PROGRAM POU
VAR
END_VAR

END_PROGRAM

(* stored: Version 1.1.0.1, ProductVersion 3.1.4024.15
   POU POU: Id {e84dcc4b-2fdc-469e-92e0-8f395adb38ff}, SpecialFunc None *)
